FUNCTION_BLOCK ResourceOld
  (* Version 1.0, 2007-08-20, Goran Cengic, Chalmers *)
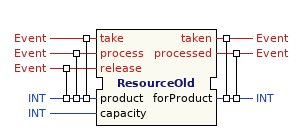
  EVENT_INPUT
    take WITH product;
    process WITH product;
    release WITH product;
  END_EVENT
  EVENT_OUTPUT
    taken WITH forProduct;
    processed WITH forProduct;
  END_EVENT
  VAR_INPUT
    product : INT;
    capacity : INT;
  END_VAR
  VAR_OUTPUT
    forProduct : INT;
  END_VAR
  VAR
    place1 : INT;
    place2 : INT;
    next : INT;
  END_VAR
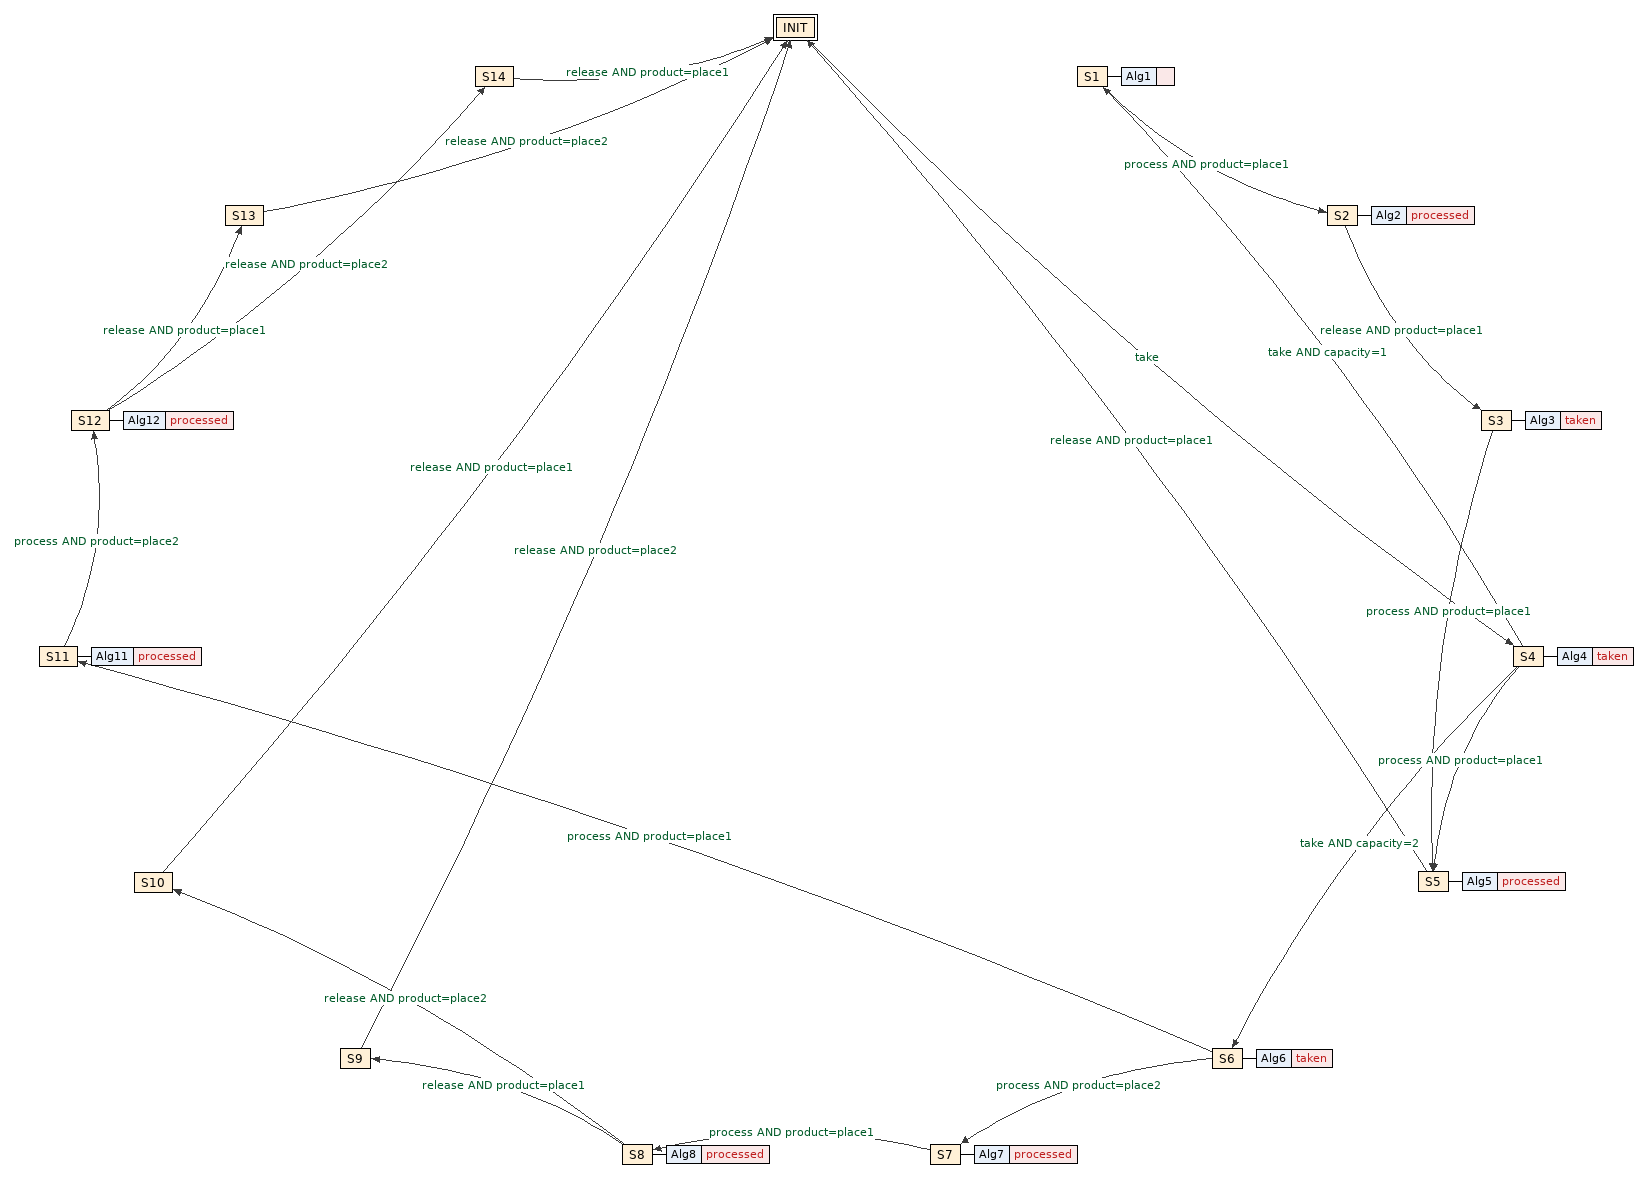
  EC_STATES
    INIT;
    S1 : Alg1;
    S2 : Alg2 -> processed;
    S3 : Alg3 -> taken;
    S4 : Alg4 -> taken;
    S5 : Alg5 -> processed;
    S6 : Alg6 -> taken;
    S7 : Alg7 -> processed;
    S8 : Alg8 -> processed;
    S9;
    S10;
    S11 : Alg11 -> processed;
    S12 : Alg12 -> processed;
    S13;
    S14;
  END_STATES
  EC_TRANSITIONS
    INIT TO S4 := take;
    S4 TO S1 := take AND capacity=1;
    S4 TO S6 := take AND capacity=2;
    S1 TO S2 := process AND product=place1;
    S2 TO S3 := release AND product=place1;
    S3 TO S5 := process AND product=place1;
    S4 TO S5 := process AND product=place1;
    S5 TO INIT := release AND product=place1;
    S6 TO S7 := process AND product=place2;
    S7 TO S8 := process AND product=place1;
    S8 TO S9 := release AND product=place1;
    S8 TO S10 := release AND product=place2;
    S9 TO INIT := release AND product=place2;
    S10 TO INIT := release AND product=place1;
    S6 TO S11 := process AND product=place1;
    S11 TO S12 := process AND product=place2;
    S12 TO S13 := release AND product=place1;
    S12 TO S14 := release AND product=place2;
    S13 TO INIT := release AND product=place2;
    S14 TO INIT := release AND product=place1;
  END_TRANSITIONS
  ALGORITHM Alg1 IN Java:
next = product;
  END_ALGORITHM
  ALGORITHM Alg2 IN Java:
forProduct = place1;
  END_ALGORITHM
  ALGORITHM Alg3 IN Java:
place1 = next; forProduct = place1;
  END_ALGORITHM
  ALGORITHM Alg4 IN Java:
place1 = product; forProduct = place1;
  END_ALGORITHM
  ALGORITHM Alg5 IN Java:
forProduct = place1;
  END_ALGORITHM
  ALGORITHM Alg6 IN Java:
place2 = product; forProduct = place2;
  END_ALGORITHM
  ALGORITHM Alg7 IN Java:
forProduct = place2;
  END_ALGORITHM
  ALGORITHM Alg8 IN Java:
forProduct = place1;
  END_ALGORITHM
  ALGORITHM Alg11 IN Java:
forProduct = place1;
  END_ALGORITHM
  ALGORITHM Alg12 IN Java:
forProduct = place2;
  END_ALGORITHM
END_FUNCTION_BLOCK
(* other elements stored in the file *)
(* <ECC> <ECState Name="INIT" /> <ECState Name="S1" > <ECAction Algorithm="PrintAlg1"/> <ECAction Algorithm="Alg1"/> </ECState> <ECState Name="S2" > <ECAction Algorithm="PrintAlg2"/> <ECAction Algorithm="Alg2" Output="processed"/> </ECState> <ECState Name="S3" > <ECAction Algorithm="PrintAlg3"/> <ECAction Algorithm="Alg3" Output="taken"/> </ECState> <ECState Name="S4" > <ECAction Algorithm="PrintAlg4"/> <ECAction Algorithm="Alg4" Output="taken"/> </ECState> <ECState Name="S5" > <ECAction Algorithm="PrintAlg5"/> <ECAction Algorithm="Alg5" Output="processed"/> </ECState> <ECState Name="S6" > <ECAction Algorithm="PrintAlg6"/> <ECAction Algorithm="Alg6" Output="taken"/> </ECState> <ECState Name="S7" > <ECAction Algorithm="PrintAlg7"/> <ECAction Algorithm="Alg7" Output="processed"/> </ECState> <ECState Name="S8" > <ECAction Algorithm="PrintAlg8"/> <ECAction Algorithm="Alg8" Output="processed"/> </ECState> <ECState Name="S9" /> <ECState Name="S10" /> <ECState Name="S11" > <ECAction Algorithm="PrintAlg11"/> <ECAction Algorithm="Alg11" Output="processed"/> </ECState> <ECState Name="S12" > <ECAction Algorithm="PrintAlg12"/> <ECAction Algorithm="Alg12" Output="processed"/> </ECState> <ECState Name="S13" /> <ECState Name="S14" /> <ECTransition Source="INIT" Destination="S4" Condition="take" /> <ECTransition Source="S4" Destination="S1" Condition="take AND capacity=1" /> <ECTransition Source="S4" Destination="S6" Condition="take AND capacity=2" /> <ECTransition Source="S1" Destination="S2" Condition="process AND product=place1" /> <ECTransition Source="S2" Destination="S3" Condition="release AND product=place1" /> <ECTransition Source="S3" Destination="S5" Condition="process AND product=place1" /> <ECTransition Source="S4" Destination="S5" Condition="process AND product=place1" /> <ECTransition Source="S5" Destination="INIT" Condition="release AND product=place1" /> <ECTransition Source="S6" Destination="S7" Condition="process AND product=place2" /> <ECTransition Source="S7" Destination="S8" Condition="process AND product=place1" /> <ECTransition Source="S8" Destination="S9" Condition="release AND product=place1" /> <ECTransition Source="S8" Destination="S10" Condition="release AND product=place2" /> <ECTransition Source="S9" Destination="INIT" Condition="release AND product=place2" /> <ECTransition Source="S10" Destination="INIT" Condition="release AND product=place1" /> <ECTransition Source="S6" Destination="S11" Condition="process AND product=place1" /> <ECTransition Source="S11" Destination="S12" Condition="process AND product=place2" /> <ECTransition Source="S12" Destination="S13" Condition="release AND product=place1" /> <ECTransition Source="S12" Destination="S14" Condition="release AND product=place2" /> <ECTransition Source="S13" Destination="INIT" Condition="release AND product=place2" /> <ECTransition Source="S14" Destination="INIT" Condition="release AND product=place1" /> </ECC> <Algorithm Name="PrintAlg1"> <Other Language="Java" Text="System.out.println(&#34;Alg1&#34;);" /> </Algorithm> <Algorithm Name="PrintAlg2"> <Other Language="Java" Text="System.out.println(&#34;Alg2&#34;);" /> </Algorithm> <Algorithm Name="PrintAlg3"> <Other Language="Java" Text="System.out.println(&#34;Alg3&#34;);" /> </Algorithm> <Algorithm Name="PrintAlg4"> <Other Language="Java" Text="System.out.println(&#34;Alg4&#34;);" /> </Algorithm> <Algorithm Name="PrintAlg5"> <Other Language="Java" Text="System.out.println(&#34;Alg5&#34;);" /> </Algorithm> <Algorithm Name="PrintAlg6"> <Other Language="Java" Text="System.out.println(&#34;Alg6&#34;);" /> </Algorithm> <Algorithm Name="PrintAlg7"> <Other Language="Java" Text="System.out.println(&#34;Alg7&#34;);" /> </Algorithm> <Algorithm Name="PrintAlg8"> <Other Language="Java" Text="System.out.println(&#34;Alg8&#34;);" /> </Algorithm> <Algorithm Name="PrintAlg11"> <Other Language="Java" Text="System.out.println(&#34;Alg11&#34;);" /> </Algorithm> <Algorithm Name="PrintAlg12"> <Other Language="Java" Text="System.out.println(&#34;Alg12&#34;);" /> </Algorithm> *)
